FUNCTION_BLOCK FB_ScaleBetween
VAR_INPUT
	RawValue : LREAL;
	RawValueMin: LREAL;
	RawValueMax : LREAL;
	ScaledValueMin : LREAL;
	ScaledValueMax : LREAL;
END_VAR
VAR_OUTPUT
	ScaledValue : LREAL;
END_VAR
VAR
END_VAR

ScaledValue :=  (((ScaledValueMax-ScaledValueMin) * (RawValue - RawValueMin)) / (RawValueMax - RawValueMin)) + ScaledValueMin;
ScaledValue := MIN(ScaledValueMax, MAX(ScaledValueMin, ScaledValue));

END_FUNCTION_BLOCK

(* stored: Version 1.1.0.1, ProductVersion 3.1.4022.16
   POU FB_ScaleBetween: Id {3f8eaedd-67fb-45e1-9633-1279513f2586}, SpecialFunc None *)
